Yaskawa INFORM job: WRREMOTE_.JBI

/JOB

//NAME WRREMOTE

//INST

///DATE 2013/06/27 10:48

///ATTR SC,RW

///GROUP1 RB1

NOP

SET I000 0

SET I002 0

SET I003 0

*LOOP

CALL JOB:WRARC IF I003=1

JUMP *LOOP IF I000>=I001

MOVL P[I002] V=I010 PL=3

INC I000

INC I002

JUMP *LOOP IF I002<32

SET I002 0

JUMP *LOOP

END
